PROGRAM P_ScopeServer
VAR

END_VAR

END_PROGRAM

(* stored: Version 1.1.0.1, ProductVersion 3.1.4026.18
   POU P_ScopeServer: Id {a56923be-0395-4c71-a7f4-1123c8bb09bb}, SpecialFunc None *)
